PROGRAM START_FORCEMEASUREMENT
VAR
	isInit : BOOL := TRUE;
	INK : INT := 1;
END_VAR

IF isInit THEN
	// Start der CAN-Sensoren
	HUB_STATE := TRUE;													// TRUE: HUB IS SENDING FRAMES, FALSE: HUS IS NOT SENDING FRAMES  	
	CAN_TRIGGER_STATE := 1;												// 1: SENSOR TRIGGER ON, 0: SENSOR TRIGGER OFF	
	CAN_CONTROL_STATE := 1;											   // SENSOR COMMANDs, 0: STOP SENSOR, 1: START SENSOR, 2: RESET SENSOR,	
	INK := INK+1 ;
END_IF

IF INK>1000 THEN
	isInit := FALSE;
	FORCE_RESET:=1;
END_IF

IF ResetForceMeasurement THEN
	CAN_CONTROL_STATE := 1;											   // SENSOR COMMANDs, 0: STOP SENSOR, 1: START SENSOR, 2: RESET SENSOR,
	ResetForceMeasurement := FALSE;
	FORCE_RESET:=1;
END_IF

END_PROGRAM

(* stored: Version 1.1.0.1, ProductVersion 3.1.4022.16
   POU START_FORCEMEASUREMENT: Id {fb953631-7e35-45d2-879f-cdb21f88fe59}, SpecialFunc None *)
